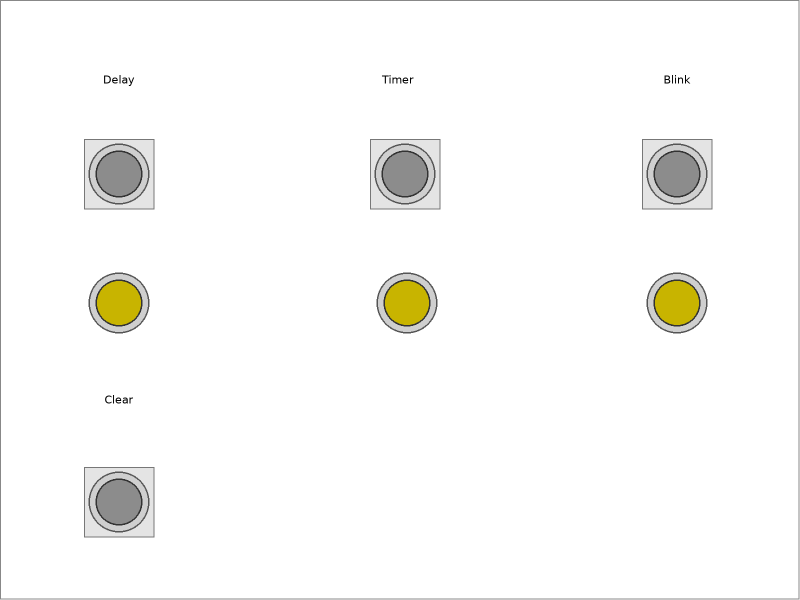
VISUALIZATION Visualization  // 800x600
    Label (44,65 150x30), "Delay"
    Label (323,65 150x30), "Timer"
    Label (602,65 150x30), "Blink"
    PushSwitch (84,139 70x70), variable: GVL.pBDelay, behaviour: TAP, style: Switch-PushSwitch-Gray
    PushSwitch (370,139 70x70), variable: GVL.pBTimer, behaviour: TAP, style: Switch-PushSwitch-Gray
    PushSwitch (642,139 70x70), variable: GVL.pBBlink, behaviour: TAP, style: Switch-PushSwitch-Gray
    Lamp1 (84,268 70x70), variable: GVL.probeDelay, style: Lamp-Lamp1-Yellow
    Lamp1 (372,268 70x70), variable: GVL.probeTimer, style: Lamp-Lamp1-Yellow
    Lamp1 (642,268 70x70), variable: GVL.probeBlink, style: Lamp-Lamp1-Yellow
    Label (44,385 150x30), "Clear"
    PushSwitch (84,467 70x70), variable: GVL.pBClear, behaviour: TAP, style: Switch-PushSwitch-Gray
END_VISUALIZATION

(* stored: Version 1.1.0.1, ProductVersion 3.1.4024.12
   Visu Visualization: Id {5151c3c8-36c0-41ee-ae39-b2ccf601b32b} *)
